# EPICS substitutions: apps/monitorApp/Db/old/caenhv_stat.substitutions
file "db/caenhv_FTOF_isOn.db"    { pattern {SEC} {1} {2} {3} {4} {5} {6} }
file "db/caenhv_FTOF_isOff.db"   { pattern {SEC} {1} {2} {3} {4} {5} {6} }
file "db/caenhv_FTOF_isComm.db"  { pattern {SEC} {1} {2} {3} {4} {5} {6} }
file "db/caenhv_FTOF_isError.db" { pattern {SEC} {1} {2} {3} {4} {5} {6} }

file "db/caenhv_ECAL_isOn.db"    { pattern {SEC} {1} {2} {3} {4} {5} {6} }
file "db/caenhv_ECAL_isOff.db"   { pattern {SEC} {1} {2} {3} {4} {5} {6} }
file "db/caenhv_ECAL_isComm.db"  { pattern {SEC} {1} {2} {3} {4} {5} {6} }
file "db/caenhv_ECAL_isError.db" { pattern {SEC} {1} {2} {3} {4} {5} {6} }

file "db/caenhv_PCAL_isOn.db"    { pattern {SEC} {1} {2} {3} {4} {5} {6} }
file "db/caenhv_PCAL_isOff.db"   { pattern {SEC} {1} {2} {3} {4} {5} {6} }
file "db/caenhv_PCAL_isComm.db"  { pattern {SEC} {1} {2} {3} {4} {5} {6} }
file "db/caenhv_PCAL_isError.db" { pattern {SEC} {1} {2} {3} {4} {5} {6} }

file "db/caenhv_LTCC_isOn.db"    { pattern {SEC} {1} {2} {3} {4} {5} {6} }
file "db/caenhv_LTCC_isOff.db"   { pattern {SEC} {1} {2} {3} {4} {5} {6} }
file "db/caenhv_LTCC_isComm.db"  { pattern {SEC} {1} {2} {3} {4} {5} {6} }
file "db/caenhv_LTCC_isError.db" { pattern {SEC} {1} {2} {3} {4} {5} {6} }

# move these to ioccaenhv_HVCTOF:
file "db/caenhv_HTCC_isOnOffComm.db" { pattern {SEC} {1} {2} {3} {4} {5} {6} }
file "db/caenhv_CTOF_isOnOffComm.db" { pattern {SEC} {1} }
